{attribute 'qualified_only'}
{attribute 'strict'}
TYPE EventCategory :
(
	Warning,
	Error,
	Transition,
	AckErr
);
END_TYPE

(* stored: Version 1.1.0.1, ProductVersion 3.1.4024.12
   DUT EventCategory: Id {27aff3ba-b6f5-4279-a9f4-15034239d504} *)
